# EPICS IOC start-up script: test/startup/st.NMX-4004-9.iocsh
#NMX pinhole changer

epicsEnvSet("MOTOR_PORT",      "$(SM_MOTOR_PORT=MCU1)")
epicsEnvSet("IPADDR",          "$(SM_IPADDR=172.30.38.65)")
epicsEnvSet("IPPORT",          "$(SM_IPPORT=48898)")
epicsEnvSet("AMSNETIDIOC",     "172.30.38.12.1.1")
epicsEnvSet("ASYN_PORT",       "$(SM_ASYN_PORT=MC_CPU1)")
epicsEnvSet("P",               "Labs-MCAG:MC-MCU-40049:")
epicsEnvSet("PREC",            "$(SM_PREC=3)")
epicsEnvSet("R",               "")
epicsEnvSet("SM_NOAXES",       "5")

epicsEnvSet("ECM_OPTIONS",     "adsPort=852;amsNetIdRemote=5.79.68.216.1.1;amsNetIdLocal=$(AMSNETIDIOC)"

# No poller yet, see ethercatmcStartPoller at the end of the script
epicsEnvSet("ECM_MOVINGPOLLPERIOD", "0")
epicsEnvSet("ECM_IDLEPOLLPERIOD", "0")
< ethercatmcController.iocsh

#
# Axis 1
#
epicsEnvSet("AXISCONFIG",      "")
epicsEnvSet("R",               "m1")
epicsEnvSet("AXIS_NO",         "$(SM_AXIS_NO=1)")
epicsEnvSet("DESC",            "$(SM_DESC=DESC)")
epicsEnvSet("EGU",             "$(SM_EGU=EGU)")
epicsEnvSet("RAWENCSTEP_ADEL", 0)
epicsEnvSet("RAWENCSTEP_MDEL", 0)
< ethercatmcActuator.iocsh

#
# Axis 2
#
epicsEnvSet("AXISCONFIG",      "")
epicsEnvSet("R",               "m2")
epicsEnvSet("AXIS_NO",         "$(SM_AXIS_NO=2)")
epicsEnvSet("DESC",            "$(SM_DESC=DESC)")
epicsEnvSet("EGU",             "$(SM_EGU=EGU)")
epicsEnvSet("RAWENCSTEP_ADEL", 0)
epicsEnvSet("RAWENCSTEP_MDEL", 0)
< ethercatmcActuator.iocsh

##
## Axis 3
##
epicsEnvSet("AXISCONFIG",      "")
epicsEnvSet("R",               "m3")
epicsEnvSet("AXIS_NO",         "$(SM_AXIS_NO=3)")
epicsEnvSet("DESC",            "$(SM_DESC=DESC)")
epicsEnvSet("EGU",             "$(SM_EGU=EGU)")
epicsEnvSet("RAWENCSTEP_ADEL", 0)
epicsEnvSet("RAWENCSTEP_MDEL", 0)
< ethercatmcIndexerAxis.iocsh
< ethercatmcAxisdebug.iocsh

#
# Axis 4
#
epicsEnvSet("AXISCONFIG",      "")
epicsEnvSet("R",               "m4")
epicsEnvSet("AXIS_NO",         "$(SM_AXIS_NO=4)")
epicsEnvSet("DESC",            "$(SM_DESC=DESC)")
epicsEnvSet("EGU",             "$(SM_EGU=EGU)")
epicsEnvSet("RAWENCSTEP_ADEL", 0)
epicsEnvSet("RAWENCSTEP_MDEL", 0)
< ethercatmcActuator.iocsh

#
# Axis 5
#
epicsEnvSet("AXISCONFIG",      "")
epicsEnvSet("R",               "m5")
epicsEnvSet("AXIS_NO",         "$(SM_AXIS_NO=5)")
epicsEnvSet("DESC",            "$(SM_DESC=DESC)")
epicsEnvSet("EGU",             "$(SM_EGU=EGU)")
epicsEnvSet("RAWENCSTEP_ADEL", 0)
epicsEnvSet("RAWENCSTEP_MDEL", 0)
< ethercatmcIndexerAxis.iocsh
< ethercatmcAxisdebug.iocsh

# Start polling, values are in millisconds
#
epicsEnvSet("MOVINGPOLLPERIOD", "200")
epicsEnvSet("IDLEPOLLPERIOD",  "500")
ethercatmcStartPoller("$(MOTOR_PORT)", "$(MOVINGPOLLPERIOD)", "$(IDLEPOLLPERIOD)")
